(* IEC 61131-3 sources: Project_Icarus/franzke_files, 5 files *)

(* ---- gvl.st ---- *)
VAR_GLOBAL

	SliderLeft			: SliderPointerFB;
	PartAtSliderL		: BOOL := FALSE;
	SliderLeftFree		: BOOL := TRUE;

	SliderRight			: SliderPointerFB;
	PartAtSliderR		: BOOL := FALSE;
	SliderRightFree		: BOOL := TRUE;

	DrillingLeft 		: DrillingMachineFB;
	PartAtDrillingL		: BOOL := FALSE;
	DrillingLeftFree	: BOOL := TRUE;

	DrillingRight		: DrillingMachineFB;
	PartAtDrillingR		: BOOL := FALSE;
	DrillingRightFree	: BOOL := TRUE;

	PartAtBeltOut		: BOOL := FALSE;
	BeltOutFree			: BOOL := TRUE;

	FaultQuitt			: BOOL;
	Fault				: BOOL;
	Warning				: BOOL;
	Info				: BOOL;

	ErrorNum			: DINT;
	ErrorButton			: BOOL;

END_VAR

(* ---- slider_pointer_fb.st ---- *)
FUNCTION_BLOCK SliderPointerFB
VAR_INPUT
	StartForward 			: BOOL := FALSE;
	StartBackward 			: BOOL := FALSE;
	pSwitchFront 	AT %I*	: BOOL;
	pSwitchBack 	AT %I*	: BOOL;
END_VAR
VAR_OUTPUT
	Busy					: BOOL := FALSE;
	Done 					: BOOL := FALSE;
	pMotorForward 	AT %Q*	: BOOL;
	pMotorBackward 	AT %Q*	: BOOL;
END_VAR
VAR
	Step 					: INT := 0;
END_VAR

CASE (Step) OF
	0 :
		IF 	(StartForward = TRUE)
		THEN
			Busy := TRUE;
			Done := FALSE;
			Step := Step + 1;
		END_IF

		IF 	(StartBackward = TRUE)
		THEN
			Busy := TRUE;
			Done := FALSE;
			Step := Step + 100;
		END_IF

	1 :
		pMotorForward := TRUE;

		IF 	(pSwitchFront = TRUE) AND
		 	(pSwitchBack = FALSE)
		THEN
			pMotorForward := FALSE;
			Step := 200; (* Handshake *)
		END_IF

	100 :
		pMotorBackward := TRUE;

		IF 	(pSwitchFront = FALSE) AND
		 	(pSwitchBack = TRUE)
		THEN
			pMotorBackward := FALSE;
			Step := 200; (* Handshake *)
		END_IF

	200 :
		Done := TRUE;

		IF	(StartForward = FALSE) AND
			(StartBackward = FALSE)
		THEN
			Busy := FALSE;
			Done := FALSE;
			Step := 0;
		END_IF

END_CASE

END_FUNCTION_BLOCK

(* ---- belt_in_manager.st ---- *)
PROGRAM BeltInManager
VAR
	Step		: DINT := 0;
	Trigger		: F_TRIG;
	WaitTimer 	: TON;
END_VAR

Trigger.CLK := SensorLoading;
Trigger();
WaitTimer.PT := T#1S;

CASE (Step) OF
	0 :
		IF (Trigger.Q = TRUE)
		THEN
			MotorBeltIn := TRUE;
			Step := Step + 1;
		END_IF

	1 :
		IF (SensorSlider1 = FALSE)
		THEN
			MotorBeltIn := FALSE;
			WaitTimer.IN := FALSE;
			WaitTimer();
			Step := Step + 1;
		END_IF

	2 :
		IF (SliderLeftFree = TRUE)
		THEN
			MotorBeltIn := TRUE;
			WaitTimer.IN := TRUE;
			WaitTimer();
			Step := Step + 1;
		END_IF

	3 :
		WaitTimer();
		IF (WaitTimer.Q = TRUE)
		THEN
			MotorBeltIn := FALSE;
			PartAtSliderL := TRUE;
			Step := Step + 1;
		END_IF

	4 :
		//Handshake to slider and reset of PartAt flag
		IF (SliderLeftFree = FALSE)
		THEN
			PartAtSliderL := FALSE;
			Step := 0;
		END_IF

END_CASE

END_PROGRAM

(* ---- drilling_manager.st ---- *)
PROGRAM DrillingManager
VAR
	First	: BOOL := TRUE;
	StepL 	: DINT := 0;
	StepR	: DINT := 0;
END_VAR

IF (First)
THEN
(*
	DrillingLeft.pMotorBelt := ADR(MotorBeltMilling);
	DrillingLeft.pMotorMachine := ADR(MotorMilling);
	DrillingLeft.pSensorMachine := ADR(SensorMilling);

	DrillingRight.pMotorBelt := ADR(MotorBeltDrilling);
	DrillingRight.pMotorMachine := ADR(MotorDrilling);
	DrillingRight.pSensorMachine := ADR(SensorDrilling);
*)
	First := FALSE;
ELSE
	DrillingLeft();
	DrillingRight();

	CASE (StepL) OF
		0 :
			DrillingLeftFree := TRUE;
			IF (PartAtDrillingL = TRUE) AND
			   (DrillingRightFree = TRUE)
			THEN
				DrillingLeftFree := FALSE;
				DrillingLeft.Start := TRUE;
				StepL := StepL + 1;
			END_IF
		1 :
			IF (DrillingLeft.Busy = TRUE) AND
			   (DrillingLeft.Done = TRUE)
			THEN
				DrillingLeft.Start := FALSE;
				PartAtDrillingR := TRUE;
				StepL := StepL + 1;
			END_IF
		2 :
			//Handshake to drilling right
			IF (DrillingRightFree = FALSE)
			THEN
				PartAtDrillingR := FALSE;
				StepL := 0;
			END_IF
	END_CASE

	CASE (StepR) OF
		0 :
			DrillingRightFree := TRUE;
			IF (PartAtDrillingR = TRUE) AND
			   (SliderRightFree = TRUE)
			THEN
				DrillingRightFree := FALSE;
				DrillingRight.Start := TRUE;
				StepR := StepR + 1;
			END_IF
		1 :
			IF (DrillingRight.Busy = TRUE) AND
			   (DrillingRight.Done = TRUE)
			THEN
				DrillingRight.Start := FALSE;
				PartAtSliderR := TRUE;
				StepR := StepR + 1;
			END_IF
		2 :
			//Handshake to slider right
			IF (SliderRightFree = FALSE)
			THEN
				PartAtSliderR := FALSE;
				StepR := 0;
			END_IF
	END_CASE

END_IF

END_PROGRAM

(* ---- plc_prg.st ---- *)
PROGRAM PLC_PRG
VAR
	WaitTimer 	: TON;
	First		: BOOL := TRUE;
END_VAR

PowerActor := TRUE;
PowerSensor := TRUE;

IF (First = TRUE)
THEN
	WaitTimer.PT := T#1S;
	WaitTimer.IN := TRUE;
	WaitTimer();
	IF (WaitTimer.Q = TRUE)
	THEN
		First := FALSE;
	END_IF
ELSE
	BeltInManager();
	SliderManager();
	DrillingManager();
	BeltOutManager();
END_IF

END_PROGRAM
